// TIA Portal V21 export
VAR_GLOBAL   // PLC tag table "KAllValvola"
END_VAR
VAR_GLOBAL CONSTANT   // user constants
   KAllValv_TimeOutPosiz : Int := 1;   // Timeout Ventilpositionierung / Valve positioning timeout / Timeout posicionamiento válvula / Délai de positionnement de la vanne / Timeout posizionamento valvola
   KAllValv_ValvolaNonInAuto : Int := 2;   // Ventil nicht in Automatik / Valve not in automatic mode / Válvula no en automático / Vanne non automatique / Valvola non in automatico
   KAllValv_ResetRichiesto : Int := 3;   // Zurücksetzen erforderlich / Reset request / Reset requerido / Réinitialisation requise / Reset richiesto
   KAllValv_ByPassFinecorsa : Int := 4;   // Bypass Endschalter / Limit switch bypass / Bypass final de carrera / Bypass de fin de course / Bypass finecorsa
   KALLValvola_05 : Int := 5;
   KALLValvola_06 : Int := 6;
   KALLValvola_07 : Int := 7;
   KALLValvola_08 : Int := 8;
   KALLValvola_09 : Int := 9;
   KALLValvola_10 : Int := 10;
   KALLValvola_11 : Int := 11;
   KALLValvola_12 : Int := 12;
   KALLValvola_13 : Int := 13;
   KALLValvola_14 : Int := 14;
   KALLValvola_15 : Int := 15;
   KALLValvola_16 : Int := 16;
END_VAR
